FUNCTION_BLOCK FB_Cylinder
VAR_INPUT
	bWorkReq			: BOOL;
	bAtHomeSensor		: BOOL;
	bAtWorkSensor		: BOOL;
	tActionDelay		: TIME := T#2S;
END_VAR
VAR_OUTPUT
	bWorkCmd			: BOOL;
	bIsAtHome			: BOOL;
	bIsAtWork			: BOOL;
	bError				: BOOL;
	sStepDiscription	: WSTRING;
END_VAR
VAR
	_step				: INT := 0;
	_timer				: TON;
END_VAR

CASE _step OF
	0	:
		sStepDiscription := "State 0 : init";
		bIsAtHome := TRUE;
		bIsAtWork := FALSE;
		bError := FALSE;	
		IF bWorkReq THEN
			_step := 1;
		END_IF
	1	:
		sStepDiscription := "State 0 : Go to work position and wait for in_position";
		bWorkCmd := TRUE;
		_timer(IN := TRUE, PT := tActionDelay);
		IF _timer.Q AND NOT bAtWorkSensor THEN
			_timer(IN := FALSE);
			_step := 99;
		END_IF
		IF bAtWorkSensor THEN
			_timer(IN := FALSE);
			_step := 2;
		END_IF
	2	:
		sStepDiscription := "State 1 : In work position";
		
END_CASE

END_FUNCTION_BLOCK

(* stored: Version 1.1.0.1, ProductVersion 3.1.4024.10
   POU FB_Cylinder: Id {f2935eea-a8fb-4477-afd0-e24e0b56f792}, SpecialFunc None *)
